(*
SPDX-FileCopyrightText: © 2026 Oleksandr Tiutyk <trofimich@gmail.com>
SPDX-License-Identifier: MIT
License: https://opensource.org/license/mit
*)

(*!
<summary>Holds namespace text initialized through the init_namespace attribute.</summary>
<description>
The compiler supplies the initial text; this block performs no runtime extraction or allocation. The owning
CurrentNamespace program exposes the stored text as borrowed metadata.
</description>
*)

FUNCTION_BLOCK INTERNAL NamespaceExtractor
VAR_OUTPUT
	//! <summary>Compiler-initialized namespace storage; consumers must not modify it.</summary>
	{attribute 'init_namespace'} 
	CurrentNamespace : STRING; 	
END_VAR

END_FUNCTION_BLOCK

(* stored: Version 1.1.0.1
   POU NamespaceExtractor: Id {0e9732c9-b183-4e43-9858-0f11c3bcf600}, SpecialFunc None *)
